FUNCTION F_GetTimeStamp : TIMESTRUCT
VAR
	fbGetTime		: GETSYSTEMTIME;	// Function Block to Fetch System Time
	TimeStamp		: T_FileTime;		// Time Stamp Structure
	Time64			: T_ULarge_Integer;	// 64-Bit Large Integer Time
	TimeShift		: LREAL;			// Amount for Time Zone Offset Shift 
	TimeZoneOffset	: DINT;				// UTC Time Zone Offset
END_VAR

// Trigger TwinCAT Function Block
fbGetTime(
	timeLoDW => Time64.dwLowPart, 
	timeHiDW => Time64.dwHighPart);

// Correct for Timezone Offset
TimeShift := DINT_TO_LREAL(ABS(TimeZoneOffset)) (*hours*) * DINT_TO_LREAL(3600) (*seconds*) * DINT_TO_LREAL(10000000) (*100ns*);

IF TimeZoneOffset < 0 THEN
	Time64 := UInt64Sub64(Time64, LREAL_TO_UINT64(TimeShift));
ELSE
	Time64 := UInt64Add64(Time64, LREAL_TO_UINT64(TimeShift));
END_IF

// Unpack Large Integer Time
TimeStamp.dwLowDateTime  := Time64.dwLowPart;
TimeStamp.dwHighDateTime := Time64.dwHighPart;

// Unpack TimeStamp to Time Structure
F_GetTimeStamp :=  FILETIME_TO_SYSTEMTIME(TimeStamp);

END_FUNCTION

(* stored: Version 1.1.0.1, ProductVersion 3.1.4024.9
   POU F_GetTimeStamp: Id {83557e2c-006f-4ccd-a1eb-a1eb60a920c5}, SpecialFunc None *)
